FUNCTION_BLOCK UnreachableState (* Basic FB with empty ECC *)
  (* Standard: 61499-2 *)
  (* Version 1.0, 2023-11-22, AK124910 *)
  PACKAGE servSeq;
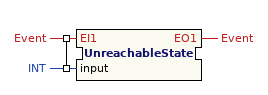
  EVENT_INPUT
    EI1 WITH input;
  END_EVENT
  EVENT_OUTPUT
    EO1;
  END_EVENT
  VAR_INPUT
    input : INT;
  END_VAR
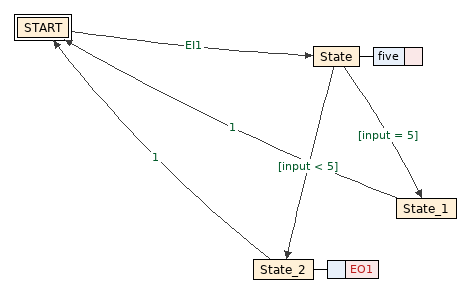
  EC_STATES
    START; (* Initial State *)
    State : five;
    State_1;
    State_2 : -> EO1;
  END_STATES
  EC_TRANSITIONS
    START TO State := EI1;
    State TO State_1 := [input = 5];
    State TO State_2 := [input < 5];
    State_2 TO START := 1;
    State_1 TO START := 1;
  END_TRANSITIONS
  ALGORITHM five IN ST:
input := 5;
  END_ALGORITHM
  (* Service external/internal_interface: Basic FB with empty ECC *)
END_FUNCTION_BLOCK
